// TIA Portal V18 export
TYPE "Runtime_Out"
   STRUCT
      TotalTime : DInt;
      TotHours : DInt;
      TotMins : DInt;
      TotSeconds : DInt;
      CurrentTime : DInt;   // Current Time in Seconds
      CurHours : DInt;
      CurMins : DInt;
      CurSeconds : DInt;
   END_STRUCT;
END_TYPE
